SUBAPPLICATION Uebung_224b_AX (* Standard IEC 61131-3 AULI_FB_CTUD (Adapter Version, ULINT) mit Terminal-Ausgabe *)
  (* Standard: 61131-3; Description: Copyright (c) 2026 Meisterschulen am Ostbahnhof This program and the accompanying materials are made available under the terms of the Eclipse Public License 2.0 which is available at https://www.eclipse.org/legal/epl-2.0/ SPDX-License-Identifier: EPL-2.0 *)
  (* Version 1.1, 2026-04-21, Franz Höpfinger, Meisterschulen am Ostbahnhof, Added terminal output for counter value *)
  (* Version 1.0, 2026-04-21, Franz Höpfinger, Meisterschulen am Ostbahnhof, initial API and implementation (Adapter version) *)
  PACKAGE Uebungen;
  IMPORT logiBUS::io::DI::logiBUS_DI::Input_I1;
  IMPORT logiBUS::io::DI::logiBUS_DI::Input_I2;
  IMPORT logiBUS::io::DI::logiBUS_DI::Input_I3;
  IMPORT logiBUS::io::DI::logiBUS_DI::Input_I4;
  IMPORT logiBUS::io::DQ::logiBUS_DO::Output_Q1;
  IMPORT logiBUS::io::DQ::logiBUS_DO::Output_Q2;
  IMPORT Uebungen::const::UT::DefaultPool_Numeric::OutputNumber_N3;
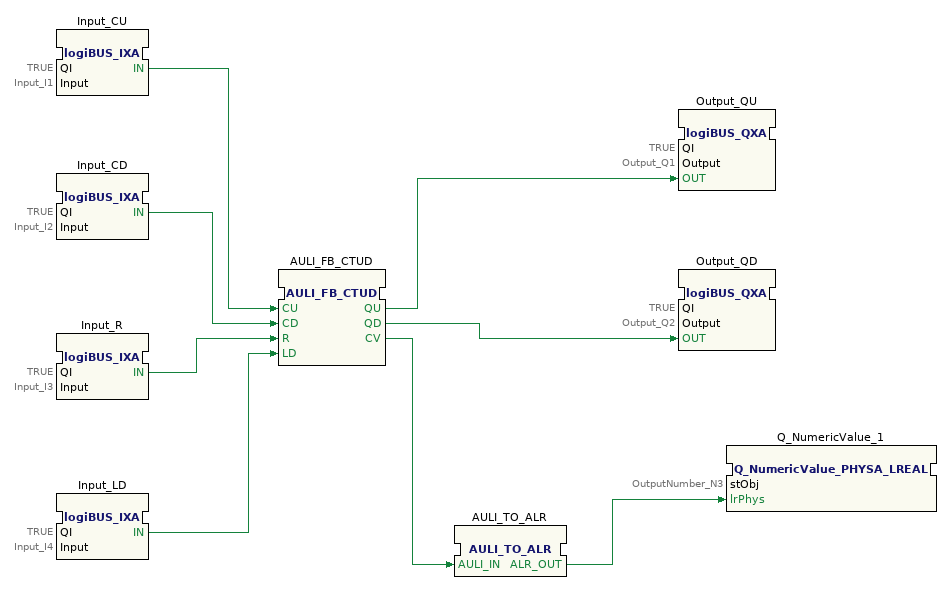
  FBS
    AULI_FB_CTUD : adapter::iec61131_3::counters::AULI_FB_CTUD;
    Input_CU : logiBUS::io::DI::logiBUS_IXA(QI := TRUE, Input := Input_I1);
    Input_CD : logiBUS::io::DI::logiBUS_IXA(QI := TRUE, Input := Input_I2);
    Input_R : logiBUS::io::DI::logiBUS_IXA(QI := TRUE, Input := Input_I3);
    Input_LD : logiBUS::io::DI::logiBUS_IXA(QI := TRUE, Input := Input_I4);
    Output_QU : logiBUS::io::DQ::logiBUS_QXA(QI := TRUE, Output := Output_Q1);
    Output_QD : logiBUS::io::DQ::logiBUS_QXA(QI := TRUE, Output := Output_Q2);
    Q_NumericValue_1 : isobus::UT::Q::Q_NumericValue_PHYSA_LREAL(stObj := OutputNumber_N3);
    AULI_TO_ALR : adapter::conversion::unidirectional::AULI_TO_ALR;
  END_FBS
  ADAPTER_CONNECTIONS
    Input_CU.IN TO AULI_FB_CTUD.CU;
    Input_CD.IN TO AULI_FB_CTUD.CD;
    Input_R.IN TO AULI_FB_CTUD.R;
    Input_LD.IN TO AULI_FB_CTUD.LD;
    AULI_FB_CTUD.QU TO Output_QU.OUT;
    AULI_FB_CTUD.QD TO Output_QD.OUT;
    AULI_FB_CTUD.CV TO AULI_TO_ALR.AULI_IN;
    AULI_TO_ALR.ALR_OUT TO Q_NumericValue_1.lrPhys;
  END_CONNECTIONS
END_SUBAPPLICATION
